(* IEC 61131-3 sources: esstee/src/tests/programs/builtins, 1 file *)

(* ---- cast.ST ---- *)
PROGRAM t

VAR
	b : BOOL;
	si : SINT;
	i : INT;
	di : DINT;
	usi : USINT;
	ui : UINT;
	udi : UDINT;
END_VAR

b := USINT_TO_BOOL(100);

END_PROGRAM
